(* CoDeSys 2.3 export: WRITE_SD_CARD.EXP *)

(* POU Write_SD_Card, FBD *)
FUNCTION_BLOCK Write_SD_Card
VAR_INPUT
	enable					: BOOL				:= FALSE;					(* enable the FUNCTION block *)
	sFileName			: STRING(30)		:= 'sdcard\plan.csv';		(* absolute path of file to operate on *)
	strData				: STRING(200)	:= '';						(* buffer for outgoing write data*)
END_VAR
VAR_OUTPUT
	done					: BOOL;
	error					: BOOL;
END_VAR
VAR
	Open_file				: FILE_Open;

	FileMode				: FILE_MODE		:= FILE_MAPPD;			(* open for write access, file stream pointer at end of the file *)
	Write_file				: FILE_Write;
	File_Handle			: CAA_HANDLE;

	close_file				: FILE_Close;

	count_closes			: CTU;
	counter_value_close	: DWORD;
	count_opened			: CTU;
	counter_value_open	: DWORD;

	zustand				: SR;
	error_open: BOOL;
	error_open_number: INT;
	error_write: BOOL;
	error_write_number: INT;
	error_close: BOOL;
	error_close_number: INT;
END_VAR
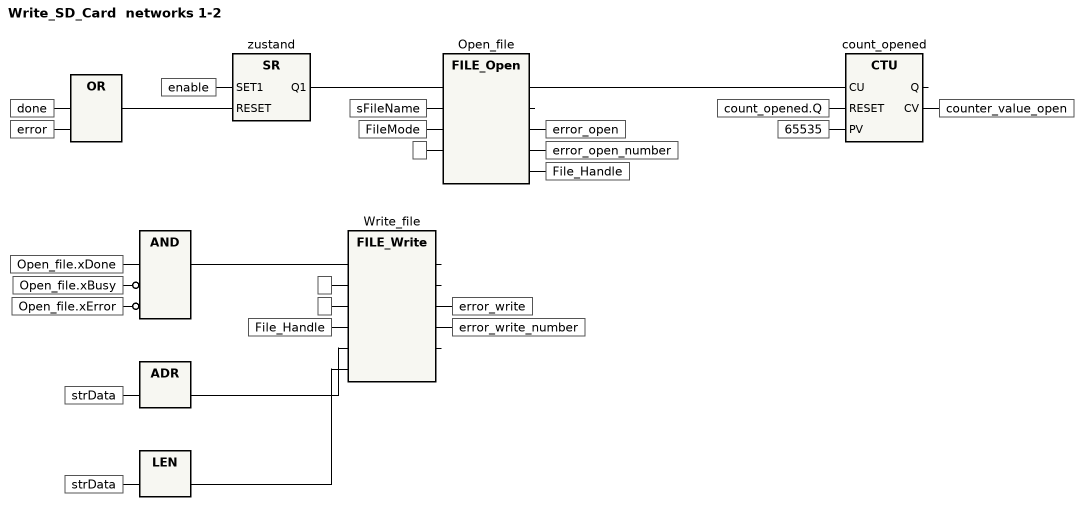
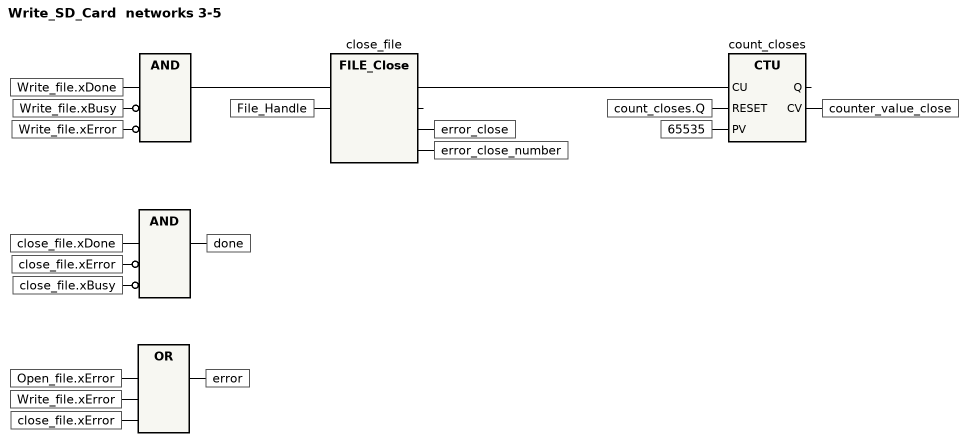
_FBD_ (* Function Block Diagram *)
NETWORK 1
	count_opened:CTU(CU: Open_file:FILE_Open(zustand:SR(SET1: enable, RESET: OR(done, error)), sFileName, FileMode, , out 3 => error_open, out 4 => error_open_number, out 5 => File_Handle), RESET: count_opened.Q, PV: 65535, CV => counter_value_open)
NETWORK 2
	Write_file:FILE_Write(AND(Open_file.xDone, NOT Open_file.xBusy, NOT Open_file.xError), , , File_Handle, ADR(strData), LEN(strData), out 3 => error_write, out 4 => error_write_number)
NETWORK 3
	count_closes:CTU(CU: close_file:FILE_Close(AND(Write_file.xDone, NOT Write_file.xBusy, NOT Write_file.xError), File_Handle, out 3 => error_close, out 4 => error_close_number), RESET: count_closes.Q, PV: 65535, CV => counter_value_close)
NETWORK 4
	AND(close_file.xDone, NOT close_file.xError, NOT close_file.xBusy) => done
NETWORK 5
	OR(Open_file.xError, Write_file.xError, close_file.xError) => error
_END_FBD_
(* the same logic as Structured Text *)
(* Network 1: see the listing above *)
(* Network 2: see the listing above *)
(* Network 3: see the listing above *)
(* Network 4 *)
done := close_file.xDone AND NOT close_file.xError AND NOT close_file.xBusy;
(* Network 5 *)
error := Open_file.xError OR Write_file.xError OR close_file.xError;
END_FUNCTION_BLOCK
